FUNCTION_BLOCK ValveControl (* Basic Function Block Type *)
  (* Standard: 61499-2 *)
  (* Version 0.0, 9/14/2008, Horst Mayer, nxtControl GmbH, Template *)
  PACKAGE Main;
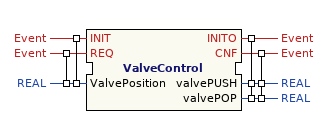
  EVENT_INPUT
    INIT WITH ValvePosition; (* Initialization Request *)
    REQ WITH ValvePosition; (* Normal Execution Request *)
  END_EVENT
  EVENT_OUTPUT
    INITO WITH valvePUSH, valvePOP; (* Initialization Confirm *)
    CNF WITH valvePUSH, valvePOP; (* Execution Confirmation *)
  END_EVENT
  VAR_INPUT
    ValvePosition : REAL;
  END_VAR
  VAR_OUTPUT
    valvePUSH : REAL;
    valvePOP : REAL;
  END_VAR
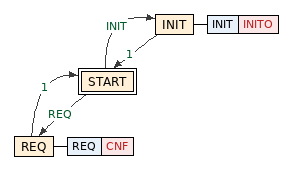
  EC_STATES
    START; (* Initial State *)
    INIT : INIT -> INITO; (* Initialization *)
    REQ : REQ -> CNF; (* Normal execution *)
  END_STATES
  EC_TRANSITIONS
    START TO INIT := INIT;
    INIT TO START := 1;
    START TO REQ := REQ;
    REQ TO START := 1;
  END_TRANSITIONS
  ALGORITHM INIT IN ST: (* Initialization algorithm *)
valvePOP := 0.0;
valvePUSH := 0.0;
  END_ALGORITHM
  ALGORITHM REQ IN ST: (* Normally executed algorithm *)
IF ValvePosition > 40 THEN
	valvePUSH := 200.0;
	valvePOP := 0.0;
ELSIF ValvePosition < 3 AND ValvePosition >=-0.5 THEN
	valvePUSH := 0.0;
	valvePOP := 200.0;
ELSIF ValvePosition = -1.0 THEN
	valvePUSH := 0.0;
	valvePOP := 0.0;
ELSE
	valvePUSH := 0.0;
	valvePOP := 0.0;
END_IF;
  END_ALGORITHM
END_FUNCTION_BLOCK
